// Mitsubishi GX Works2 project: Oil_Production_Mini_Factory   PLC: FX2N/FX2NC

PROGRAM MAIN
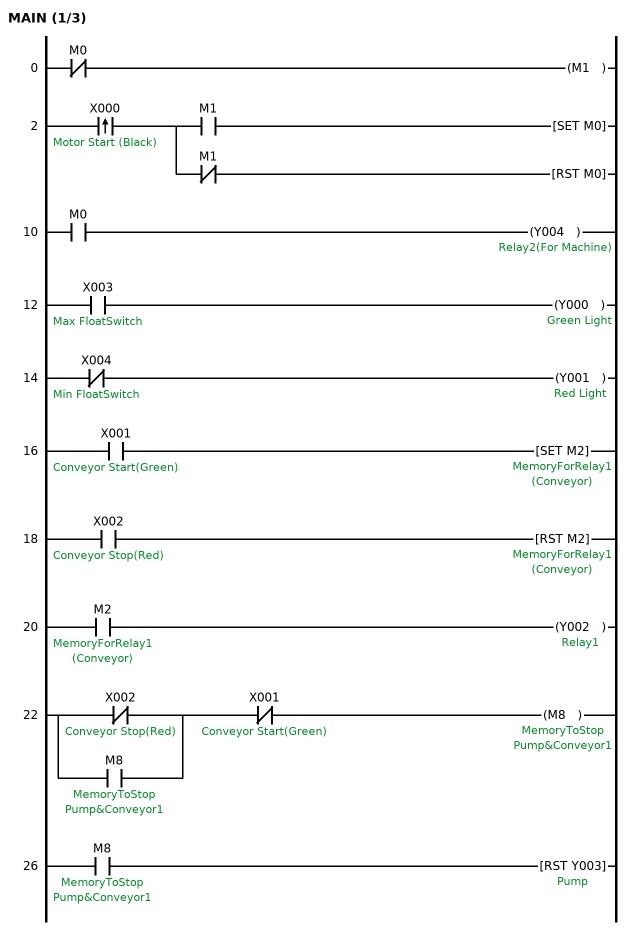
0     LDI     M0
      OUT     M1
2     LDP     X000  ; Motor Start (Black)
      MPS
      AND     M1
      SET     M0
      MPP
      ANI     M1
      RST     M0
10    LD      M0
      OUT     Y004  ; Relay2(For Machine)
12    LD      X003  ; Max FloatSwitch
      OUT     Y000  ; Green Light
14    LDI     X004  ; Min FloatSwitch
      OUT     Y001  ; Red Light
16    LD      X001  ; Conveyor Start(Green)
      SET     M2  ; MemoryForRelay1 (Conveyor)
18    LD      X002  ; Conveyor Stop(Red)
      RST     M2  ; MemoryForRelay1 (Conveyor)
20    LD      M2  ; MemoryForRelay1 (Conveyor)
      OUT     Y002  ; Relay1
22    LDI     X002  ; Conveyor Stop(Red)
      OR      M8  ; MemoryToStopPump&Conveyor1
      ANI     X001  ; Conveyor Start(Green)
      OUT     M8  ; MemoryToStopPump&Conveyor1
26    LD      M8  ; MemoryToStopPump&Conveyor1
      RST     Y003  ; Pump
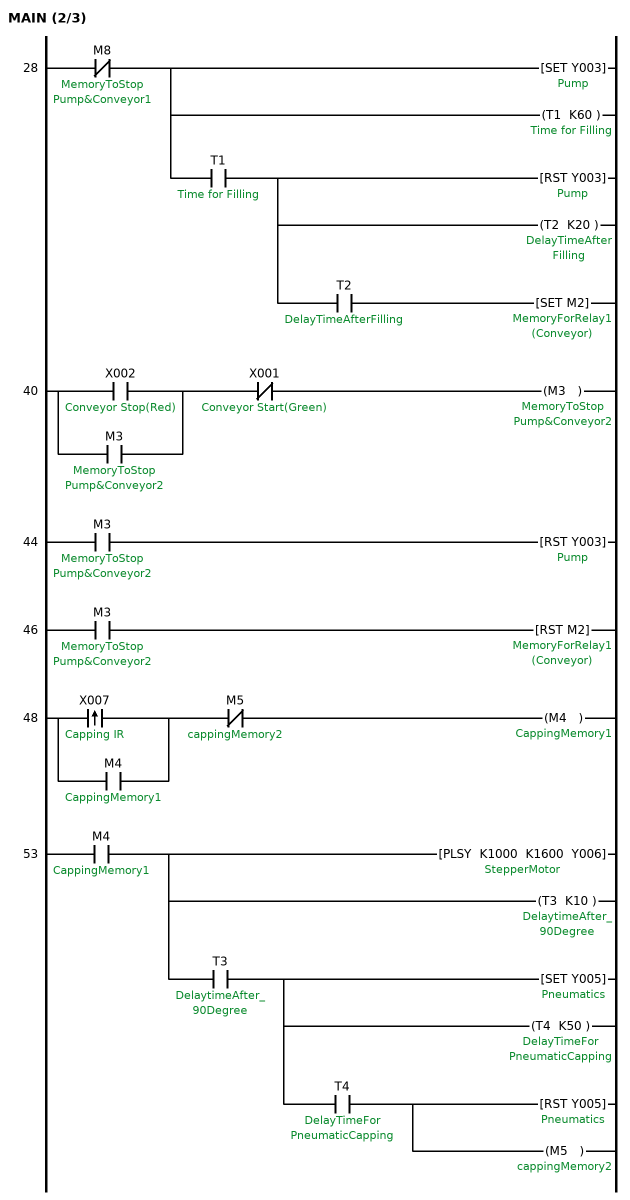
28    LDI     M8  ; MemoryToStopPump&Conveyor1
      SET     Y003  ; Pump
      OUT     T1 K60  ; Time for Filling
      AND     T1  ; Time for Filling
      RST     Y003  ; Pump
      OUT     T2 K20  ; DelayTimeAfterFilling
      AND     T2  ; DelayTimeAfterFilling
      SET     M2  ; MemoryForRelay1 (Conveyor)
40    LD      X002  ; Conveyor Stop(Red)
      OR      M3  ; MemoryToStopPump&Conveyor2
      ANI     X001  ; Conveyor Start(Green)
      OUT     M3  ; MemoryToStopPump&Conveyor2
44    LD      M3  ; MemoryToStopPump&Conveyor2
      RST     Y003  ; Pump
46    LD      M3  ; MemoryToStopPump&Conveyor2
      RST     M2  ; MemoryForRelay1 (Conveyor)
48    LDP     X007  ; Capping IR
      OR      M4  ; CappingMemory1
      ANI     M5  ; cappingMemory2
      OUT     M4  ; CappingMemory1
53    LD      M4  ; CappingMemory1
      PLSY    K1000 K1600 Y006  ; StepperMotor
      OUT     T3 K10  ; DelaytimeAfter_90Degree
      AND     T3  ; DelaytimeAfter_90Degree
      SET     Y005  ; Pneumatics
      OUT     T4 K50  ; DelayTimeForPneumaticCapping
      AND     T4  ; DelayTimeForPneumaticCapping
      RST     Y005  ; Pneumatics
      OUT     M5  ; cappingMemory2
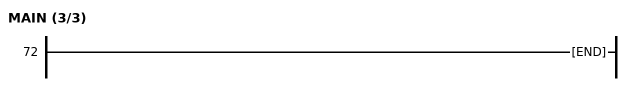
72    END
END_PROGRAM

// device comments not shown above
X005  ; filling IR
X006  ; filling IR
M7  ; MemoryForCappingIR
T0  ; Delay Before filling
